REGION Network 64: UNIT 1 STATION 3 MEASURING INITIALIZING SENSOR ALARM
   RUNG wire#powerrail
      { S7_Templates := "SrcType := Int" } EQ_Contact(in1 := "DB16006_U3_MEAS_STA_MEAS_A_CLIENT_INTERFACE".U03_FACE_A_MEAS_Read.Variable.Status, in2 := -4)
      Contact( "DB7258_UNIT_3_STA_MEAS_A_ENABLE_DISABLE".ENABLED )
      wire#w1
      Coil( "DB16000_OPC_UA_TRIGGER_ALARM".CLIENT.U3_MEAS_STA_MEAS_R.ALARMS.MEAS_INITIALIZING_SENSOR_A )
   END_RUNG
   RUNG wire#w1
      Coil( "DB426_ALARMS_WARNINGS".ALARMS.UNIT_03.FACE_R_MEASURING."724255" )
   END_RUNG
   // the same network as SCL:
   "DB16000_OPC_UA_TRIGGER_ALARM".CLIENT.U3_MEAS_STA_MEAS_R.ALARMS.MEAS_INITIALIZING_SENSOR_A := ("DB16006_U3_MEAS_STA_MEAS_A_CLIENT_INTERFACE".U03_FACE_A_MEAS_Read.Variable.Status = (-4)) AND "DB7258_UNIT_3_STA_MEAS_A_ENABLE_DISABLE".ENABLED;
   "DB426_ALARMS_WARNINGS".ALARMS.UNIT_03.FACE_R_MEASURING."724255" := "DB16000_OPC_UA_TRIGGER_ALARM".CLIENT.U3_MEAS_STA_MEAS_R.ALARMS.MEAS_INITIALIZING_SENSOR_A;
END_REGION

REGION Network 65: UNIT 3 MEASURING PLC PC MINOR VERSIONS MISMATCH WARNING
   RUNG wire#powerrail
      { S7_Templates := "SrcType := UInt" } NE_Contact(in1 := "DB16006_U3_MEAS_STA_MEAS_A_CLIENT_INTERFACE".U03_FACE_A_MEAS_Read.Variable."Version.Minor", in2 := #VERSIONS_MINOR)
      Contact( "DB7258_UNIT_3_STA_MEAS_A_ENABLE_DISABLE".ENABLED )
      wire#w1
      Coil( "DB16000_OPC_UA_TRIGGER_ALARM".CLIENT.U3_MEAS_STA_MEAS_R.ALARMS.PLC_PC_MINOR_VERSIONS_MISMATCH_W )
   END_RUNG
   RUNG wire#w1
      Coil( "DB426_ALARMS_WARNINGS".ALARMS.WARNINGS."742136" )
   END_RUNG
   // the same network as SCL:
   "DB16000_OPC_UA_TRIGGER_ALARM".CLIENT.U3_MEAS_STA_MEAS_R.ALARMS.PLC_PC_MINOR_VERSIONS_MISMATCH_W := ("DB16006_U3_MEAS_STA_MEAS_A_CLIENT_INTERFACE".U03_FACE_A_MEAS_Read.Variable."Version.Minor" <> #VERSIONS_MINOR) AND "DB7258_UNIT_3_STA_MEAS_A_ENABLE_DISABLE".ENABLED;
   "DB426_ALARMS_WARNINGS".ALARMS.WARNINGS."742136" := "DB16000_OPC_UA_TRIGGER_ALARM".CLIENT.U3_MEAS_STA_MEAS_R.ALARMS.PLC_PC_MINOR_VERSIONS_MISMATCH_W;
END_REGION

REGION Network 66: UNIT 3 MEASURING PLC PC MAJOR VERSIONS MISMATCH ALARM
   RUNG wire#powerrail
      { S7_Templates := "SrcType := UInt" } NE_Contact(in1 := "DB16006_U3_MEAS_STA_MEAS_A_CLIENT_INTERFACE".U03_FACE_A_MEAS_Read.Variable."Version.Major", in2 := #VERSIONS_MAJOR)
      wire#w1
      Contact( "DB7258_UNIT_3_STA_MEAS_A_ENABLE_DISABLE".ENABLED )
      wire#w3
      Coil( "DB16000_OPC_UA_TRIGGER_ALARM".CLIENT.U3_MEAS_STA_MEAS_R.ALARMS.PLC_PC_MAJOR_VERSIONS_MISMATCH_A )
   END_RUNG
   RUNG wire#powerrail
      Contact( "DB16000_OPC_UA_TRIGGER_ALARM".CLIENT.U3_MEAS_STA_MEAS_R.ALARMS.PLC_PC_MAJOR_VERSIONS_MISMATCH_A )
      I_Contact( "DB2120_MPP_ITC_IPC".RESET_FAULTS )
      wire#w2
      I_Contact( "DB7300_INTERLOCK_GENERAL".GENERAL_MACHINE.FROM_CELL_TO_MACHINE_GENERAL.MEAS_STA_RESET )
   END_RUNG wire#w1
   RUNG wire#w2
      I_Contact( "DB2001_MODES_GENERAL".MG_AUX_OPTIONS.AUX_BOOL[0] )
   END_RUNG wire#w1
   RUNG wire#w3
      Coil( "DB426_ALARMS_WARNINGS".ALARMS.UNIT_03.FACE_R_MEASURING."724254" )
   END_RUNG
   // the same network as SCL:
   "DB16000_OPC_UA_TRIGGER_ALARM".CLIENT.U3_MEAS_STA_MEAS_R.ALARMS.PLC_PC_MAJOR_VERSIONS_MISMATCH_A := (("DB16006_U3_MEAS_STA_MEAS_A_CLIENT_INTERFACE".U03_FACE_A_MEAS_Read.Variable."Version.Major" <> #VERSIONS_MAJOR) OR ("DB16000_OPC_UA_TRIGGER_ALARM".CLIENT.U3_MEAS_STA_MEAS_R.ALARMS.PLC_PC_MAJOR_VERSIONS_MISMATCH_A AND NOT "DB2120_MPP_ITC_IPC".RESET_FAULTS AND (NOT "DB7300_INTERLOCK_GENERAL".GENERAL_MACHINE.FROM_CELL_TO_MACHINE_GENERAL.MEAS_STA_RESET OR NOT "DB2001_MODES_GENERAL".MG_AUX_OPTIONS.AUX_BOOL[0]))) AND "DB7258_UNIT_3_STA_MEAS_A_ENABLE_DISABLE".ENABLED;
   "DB426_ALARMS_WARNINGS".ALARMS.UNIT_03.FACE_R_MEASURING."724254" := "DB16000_OPC_UA_TRIGGER_ALARM".CLIENT.U3_MEAS_STA_MEAS_R.ALARMS.PLC_PC_MAJOR_VERSIONS_MISMATCH_A;
END_REGION

REGION Network 67: IS_SEOC ALARMS
   RUNG wire#powerrail
      Contact( "M_ONE" )
      wire#w1
      I_Contact( "DB16000_OPC_UA_TRIGGER_ALARM".CLIENT.U3_MEAS_STA_MEAS_R.ALARMS.COMPUTER_CONNECTION_A )
      I_Contact( "DB16000_OPC_UA_TRIGGER_ALARM".CLIENT.U3_MEAS_STA_MEAS_R.ALARMS.COMPUTER_GET_INDEX_LIST_A )
      I_Contact( "DB16000_OPC_UA_TRIGGER_ALARM".CLIENT.U3_MEAS_STA_MEAS_R.ALARMS.COMPUTER_GET_HANDLE_LIST_A )
      I_Contact( "DB16000_OPC_UA_TRIGGER_ALARM".CLIENT.U3_MEAS_STA_MEAS_R.ALARMS.COMPUTER_GET_METHOD_LIST_A )
      I_Contact( "DB16000_OPC_UA_TRIGGER_ALARM".CLIENT.U3_MEAS_STA_MEAS_R.ALARMS.COMPUTER_RELEASE_HANDLE_LIST_A )
      I_Contact( "DB16000_OPC_UA_TRIGGER_ALARM".CLIENT.U3_MEAS_STA_MEAS_R.ALARMS.COMPUTER_RELEASE_METHOD_LIST_A )
      I_Contact( "DB16000_OPC_UA_TRIGGER_ALARM".CLIENT.U3_MEAS_STA_MEAS_R.ALARMS.COMPUTER_DISCONNECT_A )
      I_Contact( "DB16000_OPC_UA_TRIGGER_ALARM".CLIENT.U3_MEAS_STA_MEAS_R.ALARMS.MEAS_CONNECTION_A )
      I_Contact( "DB16000_OPC_UA_TRIGGER_ALARM".CLIENT.U3_MEAS_STA_MEAS_R.ALARMS.MEAS_METHOD_WORKING_BLOCKED_A )
      Not()
      Coil( #AUX_ALARMS )
   END_RUNG
   RUNG wire#w1
      I_Contact( #AUX_ALARMS )
      I_Contact( "DB16000_OPC_UA_TRIGGER_ALARM".CLIENT.U3_MEAS_STA_MEAS_R.ALARMS.CALIBRATE_CONNECTION_A )
      I_Contact( "DB16000_OPC_UA_TRIGGER_ALARM".CLIENT.U3_MEAS_STA_MEAS_R.ALARMS.CALIBRATE_METHOD_WORKING_BLOCKED_A )
      I_Contact( "DB16000_OPC_UA_TRIGGER_ALARM".CLIENT.U3_MEAS_STA_MEAS_R.ALARMS.RESET_CONNECTION_A )
      I_Contact( "DB16000_OPC_UA_TRIGGER_ALARM".CLIENT.U3_MEAS_STA_MEAS_R.ALARMS.RESET_METHOD_WORKING_BLOCKED_A )
      I_Contact( "DB16000_OPC_UA_TRIGGER_ALARM".CLIENT.U3_MEAS_STA_MEAS_R.ALARMS.READ_VAR_CONNECTION_A )
      I_Contact( "DB16000_OPC_UA_TRIGGER_ALARM".CLIENT.U3_MEAS_STA_MEAS_R.ALARMS.READ_VAR_METHOD_WORKING_BLOCKED_A )
      I_Contact( "DB16000_OPC_UA_TRIGGER_ALARM".CLIENT.U3_MEAS_STA_MEAS_R.ALARMS.DISTANCE_CALCULATION_A )
      Not()
      Move(in := #FC_NUMBER, out1 => "DB440_MACHINE_ALARM_DECODING".GLOBAL_ALARMS_MACHINE.ALARM_DECODING)
      Contact( "M_DUMMY_OFF" )
      S_Coil( "DB440_MACHINE_ALARM_DECODING".ALARMS_UNIT_3.IS_SEOC_ALARMS )
   END_RUNG
   // the same network as SCL:
   #AUX_ALARMS := NOT ("M_ONE" AND NOT "DB16000_OPC_UA_TRIGGER_ALARM".CLIENT.U3_MEAS_STA_MEAS_R.ALARMS.COMPUTER_CONNECTION_A AND NOT "DB16000_OPC_UA_TRIGGER_ALARM".CLIENT.U3_MEAS_STA_MEAS_R.ALARMS.COMPUTER_GET_INDEX_LIST_A AND NOT "DB16000_OPC_UA_TRIGGER_ALARM".CLIENT.U3_MEAS_STA_MEAS_R.ALARMS.COMPUTER_GET_HANDLE_LIST_A AND NOT "DB16000_OPC_UA_TRIGGER_ALARM".CLIENT.U3_MEAS_STA_MEAS_R.ALARMS.COMPUTER_GET_METHOD_LIST_A AND NOT "DB16000_OPC_UA_TRIGGER_ALARM".CLIENT.U3_MEAS_STA_MEAS_R.ALARMS.COMPUTER_RELEASE_HANDLE_LIST_A AND NOT "DB16000_OPC_UA_TRIGGER_ALARM".CLIENT.U3_MEAS_STA_MEAS_R.ALARMS.COMPUTER_RELEASE_METHOD_LIST_A AND NOT "DB16000_OPC_UA_TRIGGER_ALARM".CLIENT.U3_MEAS_STA_MEAS_R.ALARMS.COMPUTER_DISCONNECT_A AND NOT "DB16000_OPC_UA_TRIGGER_ALARM".CLIENT.U3_MEAS_STA_MEAS_R.ALARMS.MEAS_CONNECTION_A AND NOT "DB16000_OPC_UA_TRIGGER_ALARM".CLIENT.U3_MEAS_STA_MEAS_R.ALARMS.MEAS_METHOD_WORKING_BLOCKED_A);
   #_w1 := NOT ("M_ONE" AND NOT #AUX_ALARMS AND NOT "DB16000_OPC_UA_TRIGGER_ALARM".CLIENT.U3_MEAS_STA_MEAS_R.ALARMS.CALIBRATE_CONNECTION_A AND NOT "DB16000_OPC_UA_TRIGGER_ALARM".CLIENT.U3_MEAS_STA_MEAS_R.ALARMS.CALIBRATE_METHOD_WORKING_BLOCKED_A AND NOT "DB16000_OPC_UA_TRIGGER_ALARM".CLIENT.U3_MEAS_STA_MEAS_R.ALARMS.RESET_CONNECTION_A AND NOT "DB16000_OPC_UA_TRIGGER_ALARM".CLIENT.U3_MEAS_STA_MEAS_R.ALARMS.RESET_METHOD_WORKING_BLOCKED_A AND NOT "DB16000_OPC_UA_TRIGGER_ALARM".CLIENT.U3_MEAS_STA_MEAS_R.ALARMS.READ_VAR_CONNECTION_A AND NOT "DB16000_OPC_UA_TRIGGER_ALARM".CLIENT.U3_MEAS_STA_MEAS_R.ALARMS.READ_VAR_METHOD_WORKING_BLOCKED_A AND NOT "DB16000_OPC_UA_TRIGGER_ALARM".CLIENT.U3_MEAS_STA_MEAS_R.ALARMS.DISTANCE_CALCULATION_A);
   IF #_w1 THEN "DB440_MACHINE_ALARM_DECODING".GLOBAL_ALARMS_MACHINE.ALARM_DECODING := #FC_NUMBER; END_IF;
   IF #_w1 AND "M_DUMMY_OFF" THEN
       "DB440_MACHINE_ALARM_DECODING".ALARMS_UNIT_3.IS_SEOC_ALARMS := TRUE;
   END_IF;
END_REGION

REGION Network 68: RETURN HOME POSITION RUN OUT ALARMS
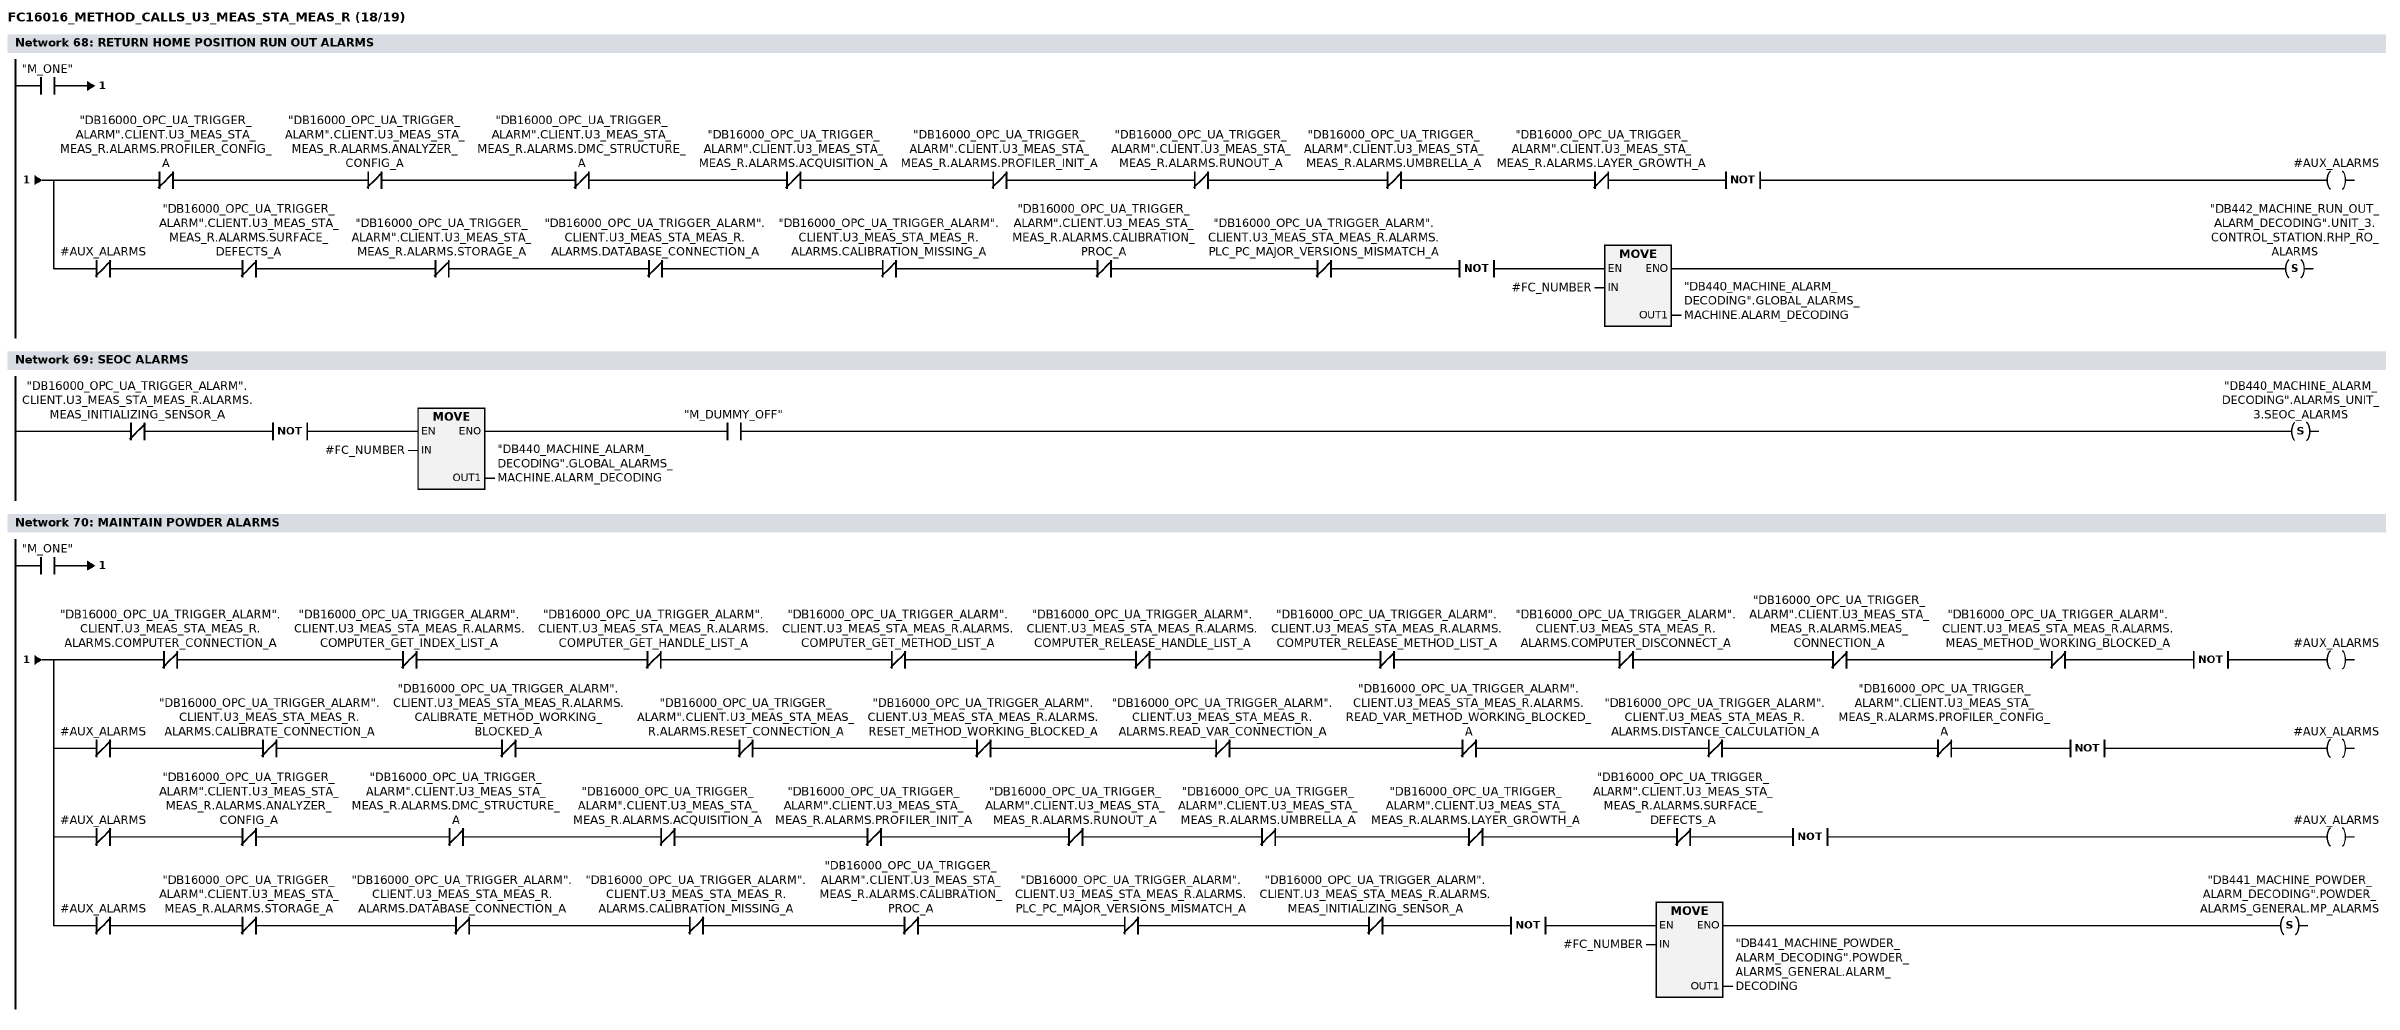
   RUNG wire#powerrail
      Contact( "M_ONE" )
      wire#w1
      I_Contact( "DB16000_OPC_UA_TRIGGER_ALARM".CLIENT.U3_MEAS_STA_MEAS_R.ALARMS.PROFILER_CONFIG_A )
      I_Contact( "DB16000_OPC_UA_TRIGGER_ALARM".CLIENT.U3_MEAS_STA_MEAS_R.ALARMS.ANALYZER_CONFIG_A )
      I_Contact( "DB16000_OPC_UA_TRIGGER_ALARM".CLIENT.U3_MEAS_STA_MEAS_R.ALARMS.DMC_STRUCTURE_A )
      I_Contact( "DB16000_OPC_UA_TRIGGER_ALARM".CLIENT.U3_MEAS_STA_MEAS_R.ALARMS.ACQUISITION_A )
      I_Contact( "DB16000_OPC_UA_TRIGGER_ALARM".CLIENT.U3_MEAS_STA_MEAS_R.ALARMS.PROFILER_INIT_A )
      I_Contact( "DB16000_OPC_UA_TRIGGER_ALARM".CLIENT.U3_MEAS_STA_MEAS_R.ALARMS.RUNOUT_A )
      I_Contact( "DB16000_OPC_UA_TRIGGER_ALARM".CLIENT.U3_MEAS_STA_MEAS_R.ALARMS.UMBRELLA_A )
      I_Contact( "DB16000_OPC_UA_TRIGGER_ALARM".CLIENT.U3_MEAS_STA_MEAS_R.ALARMS.LAYER_GROWTH_A )
      Not()
      Coil( #AUX_ALARMS )
   END_RUNG
   RUNG wire#w1
      I_Contact( #AUX_ALARMS )
      I_Contact( "DB16000_OPC_UA_TRIGGER_ALARM".CLIENT.U3_MEAS_STA_MEAS_R.ALARMS.SURFACE_DEFECTS_A )
      I_Contact( "DB16000_OPC_UA_TRIGGER_ALARM".CLIENT.U3_MEAS_STA_MEAS_R.ALARMS.STORAGE_A )
      I_Contact( "DB16000_OPC_UA_TRIGGER_ALARM".CLIENT.U3_MEAS_STA_MEAS_R.ALARMS.DATABASE_CONNECTION_A )
      I_Contact( "DB16000_OPC_UA_TRIGGER_ALARM".CLIENT.U3_MEAS_STA_MEAS_R.ALARMS.CALIBRATION_MISSING_A )
      I_Contact( "DB16000_OPC_UA_TRIGGER_ALARM".CLIENT.U3_MEAS_STA_MEAS_R.ALARMS.CALIBRATION_PROC_A )
      I_Contact( "DB16000_OPC_UA_TRIGGER_ALARM".CLIENT.U3_MEAS_STA_MEAS_R.ALARMS.PLC_PC_MAJOR_VERSIONS_MISMATCH_A )
      Not()
      Move(in := #FC_NUMBER, out1 => "DB440_MACHINE_ALARM_DECODING".GLOBAL_ALARMS_MACHINE.ALARM_DECODING)
      S_Coil( "DB442_MACHINE_RUN_OUT_ALARM_DECODING".UNIT_3.CONTROL_STATION.RHP_RO_ALARMS )
   END_RUNG
   // the same network as SCL:
   #AUX_ALARMS := NOT ("M_ONE" AND NOT "DB16000_OPC_UA_TRIGGER_ALARM".CLIENT.U3_MEAS_STA_MEAS_R.ALARMS.PROFILER_CONFIG_A AND NOT "DB16000_OPC_UA_TRIGGER_ALARM".CLIENT.U3_MEAS_STA_MEAS_R.ALARMS.ANALYZER_CONFIG_A AND NOT "DB16000_OPC_UA_TRIGGER_ALARM".CLIENT.U3_MEAS_STA_MEAS_R.ALARMS.DMC_STRUCTURE_A AND NOT "DB16000_OPC_UA_TRIGGER_ALARM".CLIENT.U3_MEAS_STA_MEAS_R.ALARMS.ACQUISITION_A AND NOT "DB16000_OPC_UA_TRIGGER_ALARM".CLIENT.U3_MEAS_STA_MEAS_R.ALARMS.PROFILER_INIT_A AND NOT "DB16000_OPC_UA_TRIGGER_ALARM".CLIENT.U3_MEAS_STA_MEAS_R.ALARMS.RUNOUT_A AND NOT "DB16000_OPC_UA_TRIGGER_ALARM".CLIENT.U3_MEAS_STA_MEAS_R.ALARMS.UMBRELLA_A AND NOT "DB16000_OPC_UA_TRIGGER_ALARM".CLIENT.U3_MEAS_STA_MEAS_R.ALARMS.LAYER_GROWTH_A);
   IF NOT ("M_ONE" AND NOT #AUX_ALARMS AND NOT "DB16000_OPC_UA_TRIGGER_ALARM".CLIENT.U3_MEAS_STA_MEAS_R.ALARMS.SURFACE_DEFECTS_A AND NOT "DB16000_OPC_UA_TRIGGER_ALARM".CLIENT.U3_MEAS_STA_MEAS_R.ALARMS.STORAGE_A AND NOT "DB16000_OPC_UA_TRIGGER_ALARM".CLIENT.U3_MEAS_STA_MEAS_R.ALARMS.DATABASE_CONNECTION_A AND NOT "DB16000_OPC_UA_TRIGGER_ALARM".CLIENT.U3_MEAS_STA_MEAS_R.ALARMS.CALIBRATION_MISSING_A AND NOT "DB16000_OPC_UA_TRIGGER_ALARM".CLIENT.U3_MEAS_STA_MEAS_R.ALARMS.CALIBRATION_PROC_A AND NOT "DB16000_OPC_UA_TRIGGER_ALARM".CLIENT.U3_MEAS_STA_MEAS_R.ALARMS.PLC_PC_MAJOR_VERSIONS_MISMATCH_A) THEN
       "DB440_MACHINE_ALARM_DECODING".GLOBAL_ALARMS_MACHINE.ALARM_DECODING := #FC_NUMBER;
       "DB442_MACHINE_RUN_OUT_ALARM_DECODING".UNIT_3.CONTROL_STATION.RHP_RO_ALARMS := TRUE;
   END_IF;
END_REGION

REGION Network 69: SEOC ALARMS
   RUNG wire#powerrail
      I_Contact( "DB16000_OPC_UA_TRIGGER_ALARM".CLIENT.U3_MEAS_STA_MEAS_R.ALARMS.MEAS_INITIALIZING_SENSOR_A )
      Not()
      Move(in := #FC_NUMBER, out1 => "DB440_MACHINE_ALARM_DECODING".GLOBAL_ALARMS_MACHINE.ALARM_DECODING)
      Contact( "M_DUMMY_OFF" )
      S_Coil( "DB440_MACHINE_ALARM_DECODING".ALARMS_UNIT_3.SEOC_ALARMS )
   END_RUNG
   // the same network as SCL:
   #_w1 := NOT (NOT "DB16000_OPC_UA_TRIGGER_ALARM".CLIENT.U3_MEAS_STA_MEAS_R.ALARMS.MEAS_INITIALIZING_SENSOR_A);
   IF #_w1 THEN "DB440_MACHINE_ALARM_DECODING".GLOBAL_ALARMS_MACHINE.ALARM_DECODING := #FC_NUMBER; END_IF;
   IF #_w1 AND "M_DUMMY_OFF" THEN "DB440_MACHINE_ALARM_DECODING".ALARMS_UNIT_3.SEOC_ALARMS := TRUE; END_IF;
END_REGION

REGION Network 70: MAINTAIN POWDER ALARMS
   RUNG wire#powerrail
      Contact( "M_ONE" )
      wire#w1
      I_Contact( "DB16000_OPC_UA_TRIGGER_ALARM".CLIENT.U3_MEAS_STA_MEAS_R.ALARMS.COMPUTER_CONNECTION_A )
      I_Contact( "DB16000_OPC_UA_TRIGGER_ALARM".CLIENT.U3_MEAS_STA_MEAS_R.ALARMS.COMPUTER_GET_INDEX_LIST_A )
      I_Contact( "DB16000_OPC_UA_TRIGGER_ALARM".CLIENT.U3_MEAS_STA_MEAS_R.ALARMS.COMPUTER_GET_HANDLE_LIST_A )
      I_Contact( "DB16000_OPC_UA_TRIGGER_ALARM".CLIENT.U3_MEAS_STA_MEAS_R.ALARMS.COMPUTER_GET_METHOD_LIST_A )
      I_Contact( "DB16000_OPC_UA_TRIGGER_ALARM".CLIENT.U3_MEAS_STA_MEAS_R.ALARMS.COMPUTER_RELEASE_HANDLE_LIST_A )
      I_Contact( "DB16000_OPC_UA_TRIGGER_ALARM".CLIENT.U3_MEAS_STA_MEAS_R.ALARMS.COMPUTER_RELEASE_METHOD_LIST_A )
      I_Contact( "DB16000_OPC_UA_TRIGGER_ALARM".CLIENT.U3_MEAS_STA_MEAS_R.ALARMS.COMPUTER_DISCONNECT_A )
      I_Contact( "DB16000_OPC_UA_TRIGGER_ALARM".CLIENT.U3_MEAS_STA_MEAS_R.ALARMS.MEAS_CONNECTION_A )
      I_Contact( "DB16000_OPC_UA_TRIGGER_ALARM".CLIENT.U3_MEAS_STA_MEAS_R.ALARMS.MEAS_METHOD_WORKING_BLOCKED_A )
      Not()
      Coil( #AUX_ALARMS )
   END_RUNG
   RUNG wire#w1
      I_Contact( #AUX_ALARMS )
      I_Contact( "DB16000_OPC_UA_TRIGGER_ALARM".CLIENT.U3_MEAS_STA_MEAS_R.ALARMS.CALIBRATE_CONNECTION_A )
      I_Contact( "DB16000_OPC_UA_TRIGGER_ALARM".CLIENT.U3_MEAS_STA_MEAS_R.ALARMS.CALIBRATE_METHOD_WORKING_BLOCKED_A )
      I_Contact( "DB16000_OPC_UA_TRIGGER_ALARM".CLIENT.U3_MEAS_STA_MEAS_R.ALARMS.RESET_CONNECTION_A )
      I_Contact( "DB16000_OPC_UA_TRIGGER_ALARM".CLIENT.U3_MEAS_STA_MEAS_R.ALARMS.RESET_METHOD_WORKING_BLOCKED_A )
      I_Contact( "DB16000_OPC_UA_TRIGGER_ALARM".CLIENT.U3_MEAS_STA_MEAS_R.ALARMS.READ_VAR_CONNECTION_A )
      I_Contact( "DB16000_OPC_UA_TRIGGER_ALARM".CLIENT.U3_MEAS_STA_MEAS_R.ALARMS.READ_VAR_METHOD_WORKING_BLOCKED_A )
      I_Contact( "DB16000_OPC_UA_TRIGGER_ALARM".CLIENT.U3_MEAS_STA_MEAS_R.ALARMS.DISTANCE_CALCULATION_A )
      I_Contact( "DB16000_OPC_UA_TRIGGER_ALARM".CLIENT.U3_MEAS_STA_MEAS_R.ALARMS.PROFILER_CONFIG_A )
      Not()
      Coil( #AUX_ALARMS )
   END_RUNG
   RUNG wire#w1
      I_Contact( #AUX_ALARMS )
      I_Contact( "DB16000_OPC_UA_TRIGGER_ALARM".CLIENT.U3_MEAS_STA_MEAS_R.ALARMS.ANALYZER_CONFIG_A )
      I_Contact( "DB16000_OPC_UA_TRIGGER_ALARM".CLIENT.U3_MEAS_STA_MEAS_R.ALARMS.DMC_STRUCTURE_A )
      I_Contact( "DB16000_OPC_UA_TRIGGER_ALARM".CLIENT.U3_MEAS_STA_MEAS_R.ALARMS.ACQUISITION_A )
      I_Contact( "DB16000_OPC_UA_TRIGGER_ALARM".CLIENT.U3_MEAS_STA_MEAS_R.ALARMS.PROFILER_INIT_A )
      I_Contact( "DB16000_OPC_UA_TRIGGER_ALARM".CLIENT.U3_MEAS_STA_MEAS_R.ALARMS.RUNOUT_A )
      I_Contact( "DB16000_OPC_UA_TRIGGER_ALARM".CLIENT.U3_MEAS_STA_MEAS_R.ALARMS.UMBRELLA_A )
      I_Contact( "DB16000_OPC_UA_TRIGGER_ALARM".CLIENT.U3_MEAS_STA_MEAS_R.ALARMS.LAYER_GROWTH_A )
      I_Contact( "DB16000_OPC_UA_TRIGGER_ALARM".CLIENT.U3_MEAS_STA_MEAS_R.ALARMS.SURFACE_DEFECTS_A )
      Not()
      Coil( #AUX_ALARMS )
   END_RUNG
   RUNG wire#w1
      I_Contact( #AUX_ALARMS )
      I_Contact( "DB16000_OPC_UA_TRIGGER_ALARM".CLIENT.U3_MEAS_STA_MEAS_R.ALARMS.STORAGE_A )
      I_Contact( "DB16000_OPC_UA_TRIGGER_ALARM".CLIENT.U3_MEAS_STA_MEAS_R.ALARMS.DATABASE_CONNECTION_A )
      I_Contact( "DB16000_OPC_UA_TRIGGER_ALARM".CLIENT.U3_MEAS_STA_MEAS_R.ALARMS.CALIBRATION_MISSING_A )
      I_Contact( "DB16000_OPC_UA_TRIGGER_ALARM".CLIENT.U3_MEAS_STA_MEAS_R.ALARMS.CALIBRATION_PROC_A )
      I_Contact( "DB16000_OPC_UA_TRIGGER_ALARM".CLIENT.U3_MEAS_STA_MEAS_R.ALARMS.PLC_PC_MAJOR_VERSIONS_MISMATCH_A )
      I_Contact( "DB16000_OPC_UA_TRIGGER_ALARM".CLIENT.U3_MEAS_STA_MEAS_R.ALARMS.MEAS_INITIALIZING_SENSOR_A )
      Not()
      Move(in := #FC_NUMBER, out1 => "DB441_MACHINE_POWDER_ALARM_DECODING".POWDER_ALARMS_GENERAL.ALARM_DECODING)
      S_Coil( "DB441_MACHINE_POWDER_ALARM_DECODING".POWDER_ALARMS_GENERAL.MP_ALARMS )
   END_RUNG
   // the same network as SCL:
   #AUX_ALARMS := NOT ("M_ONE" AND NOT "DB16000_OPC_UA_TRIGGER_ALARM".CLIENT.U3_MEAS_STA_MEAS_R.ALARMS.COMPUTER_CONNECTION_A AND NOT "DB16000_OPC_UA_TRIGGER_ALARM".CLIENT.U3_MEAS_STA_MEAS_R.ALARMS.COMPUTER_GET_INDEX_LIST_A AND NOT "DB16000_OPC_UA_TRIGGER_ALARM".CLIENT.U3_MEAS_STA_MEAS_R.ALARMS.COMPUTER_GET_HANDLE_LIST_A AND NOT "DB16000_OPC_UA_TRIGGER_ALARM".CLIENT.U3_MEAS_STA_MEAS_R.ALARMS.COMPUTER_GET_METHOD_LIST_A AND NOT "DB16000_OPC_UA_TRIGGER_ALARM".CLIENT.U3_MEAS_STA_MEAS_R.ALARMS.COMPUTER_RELEASE_HANDLE_LIST_A AND NOT "DB16000_OPC_UA_TRIGGER_ALARM".CLIENT.U3_MEAS_STA_MEAS_R.ALARMS.COMPUTER_RELEASE_METHOD_LIST_A AND NOT "DB16000_OPC_UA_TRIGGER_ALARM".CLIENT.U3_MEAS_STA_MEAS_R.ALARMS.COMPUTER_DISCONNECT_A AND NOT "DB16000_OPC_UA_TRIGGER_ALARM".CLIENT.U3_MEAS_STA_MEAS_R.ALARMS.MEAS_CONNECTION_A AND NOT "DB16000_OPC_UA_TRIGGER_ALARM".CLIENT.U3_MEAS_STA_MEAS_R.ALARMS.MEAS_METHOD_WORKING_BLOCKED_A);
   #AUX_ALARMS := NOT ("M_ONE" AND NOT #AUX_ALARMS AND NOT "DB16000_OPC_UA_TRIGGER_ALARM".CLIENT.U3_MEAS_STA_MEAS_R.ALARMS.CALIBRATE_CONNECTION_A AND NOT "DB16000_OPC_UA_TRIGGER_ALARM".CLIENT.U3_MEAS_STA_MEAS_R.ALARMS.CALIBRATE_METHOD_WORKING_BLOCKED_A AND NOT "DB16000_OPC_UA_TRIGGER_ALARM".CLIENT.U3_MEAS_STA_MEAS_R.ALARMS.RESET_CONNECTION_A AND NOT "DB16000_OPC_UA_TRIGGER_ALARM".CLIENT.U3_MEAS_STA_MEAS_R.ALARMS.RESET_METHOD_WORKING_BLOCKED_A AND NOT "DB16000_OPC_UA_TRIGGER_ALARM".CLIENT.U3_MEAS_STA_MEAS_R.ALARMS.READ_VAR_CONNECTION_A AND NOT "DB16000_OPC_UA_TRIGGER_ALARM".CLIENT.U3_MEAS_STA_MEAS_R.ALARMS.READ_VAR_METHOD_WORKING_BLOCKED_A AND NOT "DB16000_OPC_UA_TRIGGER_ALARM".CLIENT.U3_MEAS_STA_MEAS_R.ALARMS.DISTANCE_CALCULATION_A AND NOT "DB16000_OPC_UA_TRIGGER_ALARM".CLIENT.U3_MEAS_STA_MEAS_R.ALARMS.PROFILER_CONFIG_A);
   #AUX_ALARMS := NOT ("M_ONE" AND NOT #AUX_ALARMS AND NOT "DB16000_OPC_UA_TRIGGER_ALARM".CLIENT.U3_MEAS_STA_MEAS_R.ALARMS.ANALYZER_CONFIG_A AND NOT "DB16000_OPC_UA_TRIGGER_ALARM".CLIENT.U3_MEAS_STA_MEAS_R.ALARMS.DMC_STRUCTURE_A AND NOT "DB16000_OPC_UA_TRIGGER_ALARM".CLIENT.U3_MEAS_STA_MEAS_R.ALARMS.ACQUISITION_A AND NOT "DB16000_OPC_UA_TRIGGER_ALARM".CLIENT.U3_MEAS_STA_MEAS_R.ALARMS.PROFILER_INIT_A AND NOT "DB16000_OPC_UA_TRIGGER_ALARM".CLIENT.U3_MEAS_STA_MEAS_R.ALARMS.RUNOUT_A AND NOT "DB16000_OPC_UA_TRIGGER_ALARM".CLIENT.U3_MEAS_STA_MEAS_R.ALARMS.UMBRELLA_A AND NOT "DB16000_OPC_UA_TRIGGER_ALARM".CLIENT.U3_MEAS_STA_MEAS_R.ALARMS.LAYER_GROWTH_A AND NOT "DB16000_OPC_UA_TRIGGER_ALARM".CLIENT.U3_MEAS_STA_MEAS_R.ALARMS.SURFACE_DEFECTS_A);
   IF NOT ("M_ONE" AND NOT #AUX_ALARMS AND NOT "DB16000_OPC_UA_TRIGGER_ALARM".CLIENT.U3_MEAS_STA_MEAS_R.ALARMS.STORAGE_A AND NOT "DB16000_OPC_UA_TRIGGER_ALARM".CLIENT.U3_MEAS_STA_MEAS_R.ALARMS.DATABASE_CONNECTION_A AND NOT "DB16000_OPC_UA_TRIGGER_ALARM".CLIENT.U3_MEAS_STA_MEAS_R.ALARMS.CALIBRATION_MISSING_A AND NOT "DB16000_OPC_UA_TRIGGER_ALARM".CLIENT.U3_MEAS_STA_MEAS_R.ALARMS.CALIBRATION_PROC_A AND NOT "DB16000_OPC_UA_TRIGGER_ALARM".CLIENT.U3_MEAS_STA_MEAS_R.ALARMS.PLC_PC_MAJOR_VERSIONS_MISMATCH_A AND NOT "DB16000_OPC_UA_TRIGGER_ALARM".CLIENT.U3_MEAS_STA_MEAS_R.ALARMS.MEAS_INITIALIZING_SENSOR_A) THEN
       "DB441_MACHINE_POWDER_ALARM_DECODING".POWDER_ALARMS_GENERAL.ALARM_DECODING := #FC_NUMBER;
       "DB441_MACHINE_POWDER_ALARM_DECODING".POWDER_ALARMS_GENERAL.MP_ALARMS := TRUE;
   END_IF;
END_REGION

REGION Network 71: WARNINGS
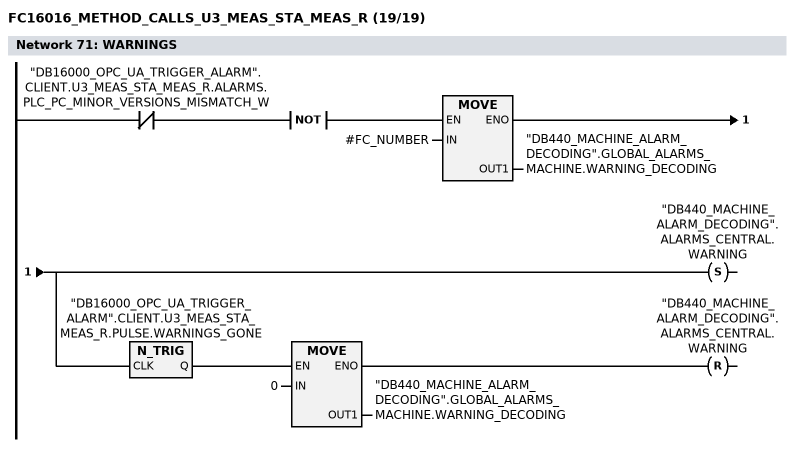
   RUNG wire#powerrail
      I_Contact( "DB16000_OPC_UA_TRIGGER_ALARM".CLIENT.U3_MEAS_STA_MEAS_R.ALARMS.PLC_PC_MINOR_VERSIONS_MISMATCH_W )
      Not()
      Move(in := #FC_NUMBER, out1 => "DB440_MACHINE_ALARM_DECODING".GLOBAL_ALARMS_MACHINE.WARNING_DECODING)
      wire#w1
      S_Coil( "DB440_MACHINE_ALARM_DECODING".ALARMS_CENTRAL.WARNING )
   END_RUNG
   RUNG wire#w1
      N_Trig( "DB16000_OPC_UA_TRIGGER_ALARM".CLIENT.U3_MEAS_STA_MEAS_R.PULSE.WARNINGS_GONE )
      Move(in := 0, out1 => "DB440_MACHINE_ALARM_DECODING".GLOBAL_ALARMS_MACHINE.WARNING_DECODING)
      R_Coil( "DB440_MACHINE_ALARM_DECODING".ALARMS_CENTRAL.WARNING )
   END_RUNG
   // the same network as SCL:
   #_w1 := NOT (NOT "DB16000_OPC_UA_TRIGGER_ALARM".CLIENT.U3_MEAS_STA_MEAS_R.ALARMS.PLC_PC_MINOR_VERSIONS_MISMATCH_W);
   IF #_w1 THEN
       "DB440_MACHINE_ALARM_DECODING".GLOBAL_ALARMS_MACHINE.WARNING_DECODING := #FC_NUMBER;
       "DB440_MACHINE_ALARM_DECODING".ALARMS_CENTRAL.WARNING := TRUE;
   END_IF;
   #_w2 := NOT #_w1 AND "DB16000_OPC_UA_TRIGGER_ALARM".CLIENT.U3_MEAS_STA_MEAS_R.PULSE.WARNINGS_GONE;   // falling edge
   "DB16000_OPC_UA_TRIGGER_ALARM".CLIENT.U3_MEAS_STA_MEAS_R.PULSE.WARNINGS_GONE := #_w1;
   IF #_w2 THEN
       "DB440_MACHINE_ALARM_DECODING".GLOBAL_ALARMS_MACHINE.WARNING_DECODING := 0;
       "DB440_MACHINE_ALARM_DECODING".ALARMS_CENTRAL.WARNING := FALSE;
   END_IF;
END_REGION
END_FUNCTION
